TYPE ST_GCR_6_0 :
(**************************************************************************************
 * 	Application		:	BoxControl Framework
 *	Revision		:	$Revision: 404529 $
 *	Revision date	:	$Date: 2018-04-23 08:21:38 +0200 (Mo., 23 Apr 2018) $
 *	Last changed by	:	$Author: b7bolm $
 *	URL				:	$URL: http://almscdc.swisslog.com/repo/SWPD/Development/BoxControlFramework/20_Release/trunk/01_Software/BCF/BCF/JumpStart/20_Product/10_App/11_Com/10_Lib/10_Conv/12_MFCS/11_SIS/01_DUTs/10_SIS_6_0/ST_GCR_6_0.TcDUT $
 *
 *	Purpose			:	GCR Structure
 *
 * ------------------------------------------------------------------------------------
 *	Copyright Swisslog [IP AG], Switzerland. All rights reserved.
 * 
 * ------------------------------------------------------------------------------------
 *	
 * 	Revision History: 
 *
 * 	VERSION			DATE			INITIALS			DESCRIPTION
 *	0.1				01.01.2001		swl					Example
 *
 **************************************************************************************)
STRUCT
	GroupName		: STRING(SIS_6_0.POSITION_STRINGLENGTH); // 12 Digit SIS Group Name MM-GGG-0000-000 
	Code			: STRING(SIS_6_0.CONTROLCODE_STRINGLENGTH); // 2 Digit Control code 
	Variable		: STRING(SIS_6_0.CONTROLVARIABLE_STRINGLENGTH); // 4 DigitControl code variable 
	ReturnCode		: STRING(SIS_6_0.ERRORCODE_STRINGLENGTH); // 4 Digit Return Code 
END_STRUCT
END_TYPE

(* stored: Version 1.1.0.1, ProductVersion 3.1.4022.12
   DUT ST_GCR_6_0: Id {42aea4df-9b21-4241-a853-20fbfbaf42dd} *)
